ABB RobotStudio station: carsuspension.rspag

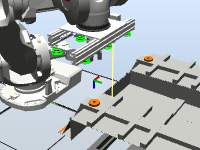
--- station ---
Station Car Suspension Ankit (saved by RobotStudio format 3)
Controller IRB_7600_340kg_2.80m
  mechanical unit ROB_1: IRB7600_340_280__01, 6 joints, base frame (0, 0, 0) mm
Layout (positions relative to the parent item):
  - IRB7600_340_280__01 [mechanism, from Robots\IRB7600_340_280_G_01.rslib] at (0, 0, 0) mm; joint values [1.0218, 0.5447, -0.711, 0.0026, 1.7386, 1.0222] (rad or m)
  - Part_10 [part, from Libraries\Part_10.rslib] at (-59.02, 745.49, 644.22) mm
  - SC_LaserSensor [smart component, from Libraries\SC_LaserSensor.rslib] at (1161.79, 1900.33, 1828.31) mm, rotated rx 180 ry -0.17 rz -180 deg
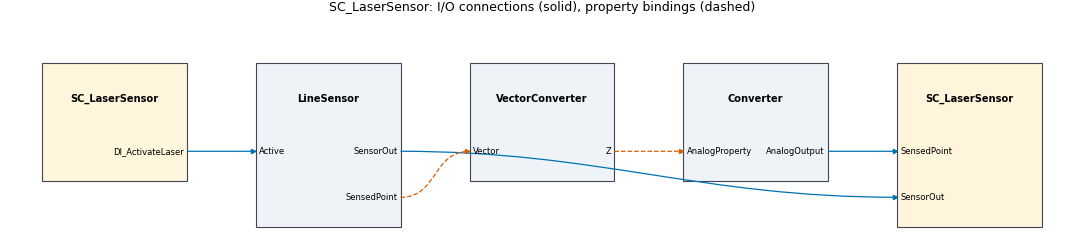
      connections:
        Converter.AnalogOutput -> SC_LaserSensor.SensedPoint
        LineSensor.SensorOut -> SC_LaserSensor.SensorOut
        SC_LaserSensor.DI_ActivateLaserSensor -> LineSensor.Active
        LineSensor.SensedPoint => VectorConverter.Vector
        VectorConverter.Z => Converter.AnalogProperty
    - LineSensor [smart component, from Components\LineSensor.rslib]
        properties: Start=[0.21 0.042 0.118]; End=[0.21 0.042 1]; Radius=1E-05; SensedPart=Car Underbody; SensedPoint=[0.949731506347656 1.94757446289063 1.11697045898437]
      - _sensorPart_ [part]
    - VectorConverter [smart component, from Components\VectorConverter.rslib]
        properties: X=0.949731506347656; Y=1.94757446289063; Z=1.11697045898437; Vector=[0.949731506347656 1.94757446289063 1.11697045898437]
    - Converter [smart component, from Components\Converter.rslib]
        properties: AnalogProperty=1.11697045898437; DigitalProperty=0; BooleanProperty=false; GroupProperty=0
  - table [part, from Libraries\table.rslib] at (1974.44, -431.38, 670) mm
  - Car Underbody [part] at (0, -200, 0) mm
  - SC_Gripper [smart component, from Libraries\SC_Gripper.rslib] at (-1443.39, 1900.33, 2562.23) mm, rotated rx 0 ry 60.17 rz 0 deg
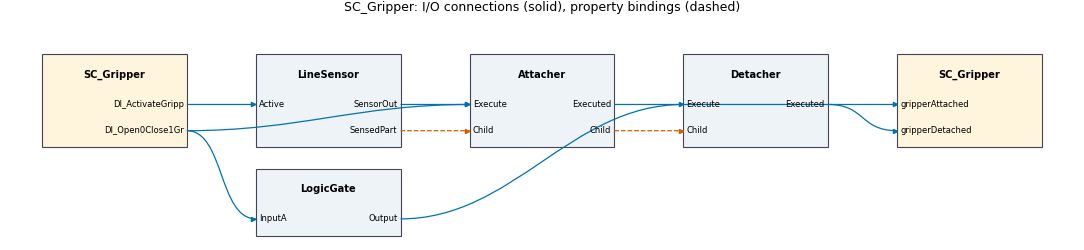
      connections:
        Attacher.Executed -> SC_Gripper.gripperAttached
        Detacher.Executed -> SC_Gripper.gripperDetached
        SC_Gripper.DI_ActivateGripper -> LineSensor.Active
        SC_Gripper.DI_Open0Close1Gripper -> Attacher.Execute
        LogicGate.Output -> Detacher.Execute
        SC_Gripper.DI_Open0Close1Gripper -> LogicGate.InputA
        LineSensor.SensorOut -> Attacher.Execute
        LineSensor.SensedPart => Attacher.Child
        Attacher.Child => Detacher.Child
    - Tool [graphiccomponentgroup, from Libraries\SC_Gripper.rslib] at (1932.51, 0, 1895) mm, rotated rx 180 ry 60 rz 180 deg
      - Vakuumgreifer [part, from Libraries\SC_Gripper.rslib]
      - GripperCylinder [part, from Libraries\SC_Gripper.rslib] at (0, 0, 85) mm
      - GripperFinger_1 [part, from Libraries\SC_Gripper.rslib] at (0, 0, 85) mm
      - GripperFinger_2 [part, from Libraries\SC_Gripper.rslib] at (0, 0, 85) mm, rotated rx 0 ry 0 rz 120 deg
      - GripperFinger_3 [part, from Libraries\SC_Gripper.rslib] at (0, 0, 85) mm, rotated rx 0 ry 0 rz -120 deg
    - LineSensor [smart component, from Components\LineSensor.rslib] at (1932.51, 0, 1895) mm, rotated rx 180 ry 60 rz 180 deg
        properties: Start=[0 0 0.215]; End=[0 0 0.225]; Radius=0.002; SensedPart=(none); SensedPoint=[1.29166296386719 1.83559130859375 1.60463647460938]
      - _sensorPart_ [part]
    - Attacher [smart component, from Components\Attacher.rslib]
        properties: Parent=Tool; Flange=0; Child=(none); Mount=false; Offset=[0 0 0]; Orientation=[0 0 0]
    - Detacher [smart component, from Components\Detacher.rslib]
        properties: Child=(none); KeepPosition=true
    - LogicGate [smart component, from Components\LogicGate.rslib]
        properties: Operator=NOT; Delay=0
  - Suspension_1 [graphiccomponentgroup, from Libraries\Suspension_1.rslib] at (2202.04, -555.68, 886.13) mm, rotated rx 180 ry 0 rz 0 deg
    - Part_4 [part, from Libraries\Suspension_1.rslib] at (0, 0, -2.49) mm
    - Part_5 [part, from Libraries\Suspension_1.rslib] at (0, 0, -2.05) mm
    - Part_6 [part, from Libraries\Suspension_1.rslib] at (0, 0, -2.05) mm
    - Part_3 [part, from Libraries\Suspension_1.rslib] at (-15.42, 2.83, 157.95) mm, rotated rx -180 ry 0 rz 0 deg
    - Part_7 [part, from Libraries\Suspension_1.rslib] at (15.59, 56.96, 120.72) mm, rotated rx -90 ry 0 rz -90 deg
  - Suspension_2 [graphiccomponentgroup, from Libraries\Suspension_2.rslib] at (2476.35, -555.68, 886.13) mm, rotated rx 180 ry 0 rz 0 deg
    - Part_4 [part, from Libraries\Suspension_2.rslib]
    - Part_5 [part, from Libraries\Suspension_2.rslib]
    - Part_6 [part, from Libraries\Suspension_2.rslib]
    - Part_3 [part, from Libraries\Suspension_2.rslib] at (-15.42, 2.83, 160) mm, rotated rx 180 ry 0 rz 0 deg
    - Part_7 [part, from Libraries\Suspension_2.rslib] at (15.59, 56.96, 122.77) mm, rotated rx -90 ry 0 rz -90 deg
Attachment: LineSensor is attached to Tool
Attachment: SC_Gripper is attached to IRB7600_340_280__01 / Link7
Attachment: Tool is attached to IRB7600_340_280__01 / Link7
Attachment: SC_LaserSensor is attached to IRB7600_340_280__01 / Link7
Attachment: Part_5 is attached to Part_4
Attachment: Part_6 is attached to Part_4
Attachment: Part_3 is attached to Part_4
Attachment: Part_7 is attached to Part_4
Attachment: Part_5 is attached to Part_4
Attachment: Part_6 is attached to Part_4
Attachment: Part_3 is attached to Part_4
Attachment: Part_7 is attached to Part_4
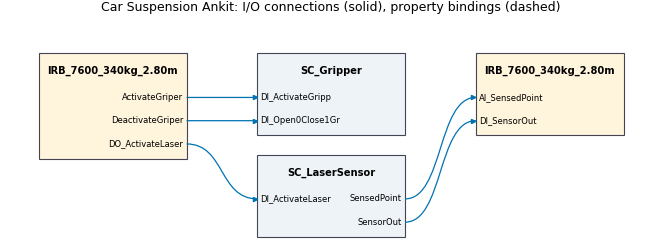
Station logic (signal -> signal, property => property):
  IRB_7600_340kg_2.80m.ActivateGriper -> SC_Gripper.DI_ActivateGripper
  IRB_7600_340kg_2.80m.DeactivateGriper -> SC_Gripper.DI_Open0Close1Gripper
  IRB_7600_340kg_2.80m.DO_ActivateLaserSensor -> SC_LaserSensor.DI_ActivateLaserSensor
  SC_LaserSensor.SensedPoint -> IRB_7600_340kg_2.80m.AI_SensedPoint
  SC_LaserSensor.SensorOut -> IRB_7600_340kg_2.80m.DI_SensorOut

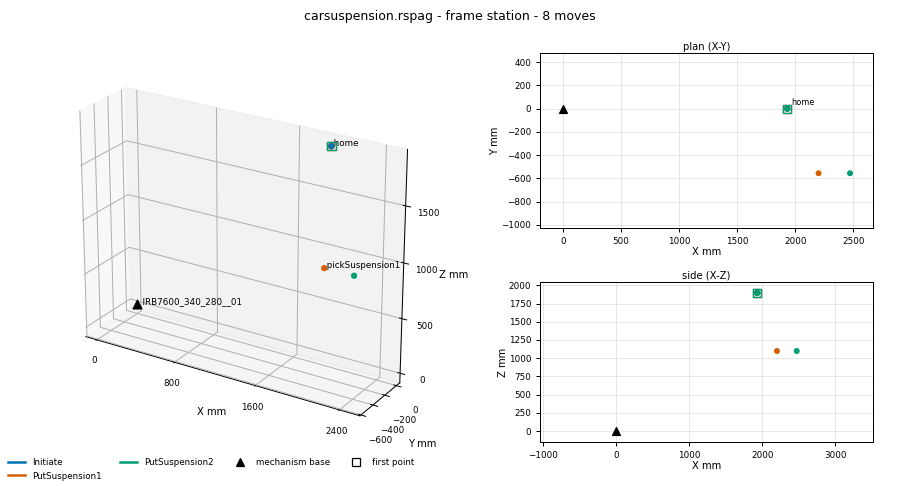
[picture p0: tool path of carsuspension.rspag in frame station, 8 of 38 moves have a stored position in this frame; points joined in program order, loops and branches not executed]
--- Backups/IRB_7600_340kg_2.80m/RAPID/TASK1/PROGMOD/CalibData.mod ---
MODULE CalibData
	TASK PERS tooldata myTool:=[TRUE,[[3.16,-2.44,456.26],[1,0,0,0]],[1,[0,0,1],[1,0,0,0],0,0,0]];
ENDMODULE

--- Backups/IRB_7600_340kg_2.80m/RAPID/TASK1/PROGMOD/Module1.mod ---
MODULE Module1
	CONST robtarget home:=[[1932.506319322,0,1894.999945226],[0.49999989,0,0.866025467,0],[0,0,0,0],[9E9,9E9,9E9,9E9,9E9,9E9]];
    CONST robtarget ScanFrontEdge:=[[201.51139568,1303.367736815,1894.998776679],[0.001498958,0.000001029,-0.999998877,0.000000047],[0,0,0,0],[9E9,9E9,9E9,9E9,9E9,9E9]];
    CONST robtarget pickSuspension1:=[[2201.608028845,-556.557878581,1098.980316128],[0.00023706,0.000000161,0.999999972,-0.00000152],[-1,0,-1,0],[9E9,9E9,9E9,9E9,9E9,9E9]];
    CONST robtarget pickSuspension2:=[[2472.738052401,-556.55975729,1098.980699702],[0.000237163,0.000000677,0.999999972,-0.000001447],[-1,0,-1,0],[9E9,9E9,9E9,9E9,9E9,9E9]];


    CONST num tcpYoffs:=42;
    CONST num tcpXoffs:=214.002;
    VAR robtarget Safehight;
    VAR robtarget next_target;
    VAR robtarget FrontEdge;
    VAR robtarget LeftEdge;
    VAR robtarget Centrep;
    VAR num HoleOffs;
    VAR robtarget CentrePoint1;
    VAR robtarget CentrePoint2;
    VAR robtarget CentrePoint3;
    VAR num Offsetz;
    VAR speeddata fast_speed:= v1000;
    VAR speeddata moderate_speed:= v500;


    PROC Initiate()
	    MoveJ home,fast_speed,z100,myTool\WObj:=wobj0;
        SetDO ActivateGriper,0;
        SetDO ActivateGriper,0;
        setdo DO_ActivateLaserSensor,0;
        Waitrob\InPos;
        WaitTime 1;
	ENDPROC

    PROC FrontEdge1()
        SetDO DO_ActivateLaserSensor,1;
        next_target:=ScanFrontEdge;

        MoveJ next_target,fast_speed,fine,tool0\WObj:=wobj0;
        WaitRob\InPos;
        WaitTime 1;
        WHILE TRUE DO
            IF  DI_SensorOut = 0 THEN
                next_target:=offs(next_target,0,100,0);
                MoveL next_target,fast_speed,fine,tool0\WObj:=wobj0;
                WaitRob\InPos;
                WaitTime 1;
            ELSE
                RETURN;
            ENDIF
        ENDWHILE
    ENDPROC
        PROC FrontEdge2()
            WHILE TRUE DO
                IF  DI_SensorOut = 1 THEN
                next_target:=Offs(next_target,0,-50,0);
                MoveL next_target,fast_speed,fine,tool0\WObj:=wobj0;
                WaitRob\InPos;
                WaitTime 0.1;
            ELSE
                FrontEdge:=next_target;
                RETURN;
                ENDIF
            ENDWHILE
        ENDPROC

         PROC FrontEdge3()
            WHILE TRUE DO
                IF  DI_SensorOut = 0 THEN
                next_target:=Offs(next_target,0,10,0);
                MoveL next_target,fast_speed,fine,tool0\WObj:=wobj0;
                WaitRob\InPos;
                WaitTime 0.1;
            ELSE
                FrontEdge:=next_target;
                RETURN;
                ENDIF
            ENDWHILE
        ENDPROC

         PROC FrontEdge4()
            WHILE TRUE DO
                IF  DI_SensorOut = 1 THEN
                next_target:=Offs(next_target,0,-1,0);
                MoveL next_target,fast_speed,fine,tool0\WObj:=wobj0;
                WaitRob\InPos;
                WaitTime 0.1;
            ELSE
                FrontEdge:=next_target;
                RETURN;
                ENDIF
            ENDWHILE
        ENDPROC

           PROC FrontEdge5()
            WHILE TRUE DO
                IF  DI_SensorOut = 0 THEN
                next_target:=Offs(next_target,0,0.1,0);
                MoveL next_target,fast_speed,fine,tool0\WObj:=wobj0;
                WaitRob\InPos;
                WaitTime 0.1;
            ELSE
                FrontEdge:=next_target;
                RETURN;
                ENDIF
            ENDWHILE
        ENDPROC

        PROC LeftEdge1()
            next_target:=Offs(FrontEdge,0,20,0);
            MoveL next_target,fast_speed,fine,tool0\WObj:=wobj0;
            WHILE TRUE DO
            IF   DI_SensorOut  = 1 THEN
                next_target:=Offs(next_target,-100,0,0);
                MoveL next_target,fast_speed,fine,tool0\WObj:=wobj0;
                WaitRob\InPos;
                WaitTime 0.5;
            ELSE
                RETURN;
            ENDIF
            ENDWHILE
        endproc
            PROC LeftEdge2()
                WHILE TRUE DO
                IF   DI_SensorOut  = 0 THEN
                next_target:=Offs(next_target,50,0,0);
                MoveL next_target,fast_speed,fine,tool0\WObj:=wobj0;
                ELSE
                LeftEdge:=Offs(next_target,-tcpXoffs,tcpYoffs,0);
                RETURN;
            ENDIF
                ENDWHILE
            ENDPROC

            PROC LeftEdge3()
                WHILE TRUE DO
                IF   DI_SensorOut  = 1 THEN
                next_target:=Offs(next_target,-10,0,0);
                MoveL next_target,fast_speed,fine,tool0\WObj:=wobj0;
                ELSE
                LeftEdge:=Offs(next_target,-tcpXoffs,tcpYoffs,0);
                RETURN;
            ENDIF
                ENDWHILE
            ENDPROC

             PROC LeftEdge4()
                WHILE TRUE DO
                IF   DI_SensorOut  = 0 THEN
                next_target:=Offs(next_target,1,0,0);
                MoveL next_target,fast_speed,fine,tool0\WObj:=wobj0;
                ELSE
                LeftEdge:=Offs(next_target,-tcpXoffs,tcpYoffs,0);
                RETURN;
            ENDIF
                ENDWHILE
            ENDPROC

             PROC LeftEdge5()
                WHILE TRUE DO
                IF   DI_SensorOut  = 1 THEN
                next_target:=Offs(next_target,-0.1,0,0);
                MoveL next_target,fast_speed,fine,tool0\WObj:=wobj0;
                ELSE
                LeftEdge:=Offs(next_target,-tcpXoffs,tcpYoffs,0);
                RETURN;
            ENDIF
                ENDWHILE
            ENDPROC


            PROC CentrePoint11()
                next_target:=Offs(next_target,220,150,0);
                MoveL next_target,fast_speed,fine,tool0\WObj:=wobj0;
                WHILE TRUE DO
                    IF  DI_SensorOut=1 THEN
                        next_target:=Offs(next_target,0,1,0);
                        MoveL next_target,fast_speed,fine,tool0\WObj:=wobj0;
                        WaitRob\InPos;
                        WaitTime 0.1;
                    ELSE
                        RETURN;
                    ENDIF
                ENDWHILE
            ENDPROC
            PROC CentrePoint12()
                 WHILE TRUE DO
                    IF  DI_SensorOut=0 THEN
                        next_target:=Offs(next_target,0,-0.1,0);
                        MoveL next_target,fast_speed,fine,tool0\WObj:=wobj0;
                        WaitRob\InPos;
                        WaitTime 0.1;
                    ELSE

                        CentrePoint1:=next_target;
                        RETURN;
                    ENDIF
                ENDWHILE
            ENDPROC
            PROC CentrePoint21()
                next_target:=Offs(next_target,0,1,0);
                MoveL next_target,fast_speed,fine,tool0\WObj:=wobj0;
                 WHILE TRUE DO
                    IF DI_Sensorout=0 THEN
                        next_target:=Offs(next_target,0,1,0);
                        MoveL next_target,fast_speed,fine,tool0\WObj:=wobj0;

                        WaitTime 1;
                    ELSE
                        Offsetz:=ai_Sensedpoint*1000;
                        RETURN;
                    ENDIF
                ENDWHILE
            ENDPROC
            PROC CentrePoint22()
                 WHILE TRUE DO
                    IF  DI_SensorOut=1 THEN
                        next_target:=Offs(next_target,0,-0.1,0);
                        MoveL next_target,fast_speed,fine,tool0\WObj:=wobj0;
                        WaitRob\InPos;
                        WaitTime 0.1;
                    ELSE

                        CentrePoint2:=next_target;
                        RETURN;
                    ENDIF
                ENDWHILE
            ENDPROC
            PROC CentrePoint31()
                 WHILE TRUE DO
                    IF  DI_SensorOut=0 THEN
                        next_target:=Offs(next_target,1,0,0);
                        MoveL next_target,fast_speed,fine,tool0\WObj:=wobj0;
                        WaitRob\InPos;
                        WaitTime 0.1;
                    ELSE
                        RETURN;
                    ENDIF
                ENDWHILE
            ENDPROC
            PROC CentrePoint32()
                 WHILE TRUE DO
                    IF  DI_SensorOut=1 THEN
                        next_target:=Offs(next_target,-0.1,0,0);
                        MoveL next_target,fast_speed,fine,tool0\WObj:=wobj0;
                        WaitRob\InPos;
                        WaitTime 0.1;
                    ELSE
                        CentrePoint3:=next_target;
                        RETURN;
                    ENDIF
                ENDWHILE
            ENDPROC
            PROC Centre()
                CentrePoint11;
                CentrePoint12;
                CentrePoint21;
                CentrePoint22;
                CentrePoint31;
                CentrePoint32;
                Centrep.trans.x:=(CentrePoint3.trans.x+CentrePoint1.trans.x)/2-tcpXoffs;
                Centrep.trans.y:=(CentrePoint3.trans.y+CentrePoint1.trans.y)/2+tcpYoffs;
                Centrep.trans.z:=Offsetz;
                Centrep.robconf:=CentrePoint3.robconf;
                Centrep.rot:=CentrePoint3.rot;
                Centrep.extax:=CentrePoint3.extax;
            ENDPROC

            PROC PutSuspension1()
                MoveL Home,fast_speed,fine,tool0\WObj:=wobj0;
                SafeHight:=Offs(pickSuspension1,0,0,500);
                MoveL Safehight,fast_speed,fine,tool0\WObj:=wobj0;
                MoveL pickSuspension1,fast_speed,fine,tool0\WObj:=wobj0;
                Setdo ActivateGriper,1;
                SetDO DeactivateGriper,1;
                WaitRob\InPos;
                WaitTime 0.5;
                MoveL Safehight,fast_speed,fine,tool0\WObj:=wobj0;
                MoveL Home,fast_speed,fine,tool0\WObj:=wobj0;
                Safehight:=offs(Centrep,0,0,250);
                MoveL Safehight,fast_speed,fine,myTool;
                MoveL Centrep,moderate_speed,fine,myTool;

                WaitRob\ZeroSpeed;
                 SetDO DeactivateGriper,0;
                MoveL Safehight,fast_speed,fine,myTool;
                SetDO ActivateGriper,0;
            ENDPROC

             PROC PutSuspension2()
                HoleOffs:=1430-(Centrep.trans.x-LeftEdge.trans.x)*2;
                MoveL Home,fast_speed,fine,tool0\WObj:=wobj0;
                Safehight:=Offs(pickSuspension2,0,0,200);
                MoveL Safehight,fast_speed,fine,tool0\WObj:=wobj0;
                MoveL pickSuspension2,fast_speed,fine,tool0\WObj:=wobj0;
                SetDO ActivateGriper,1;
                Setdo DeactivateGriper,1;
                WaitRob\InPos;
                WaitTime 0.5;
                MoveL Safehight,fast_speed,fine,tool0\WObj:=wobj0;
                SetDO ActivateGriper,0;
                MoveL Home,fast_speed,fine,tool0\WObj:=wobj0;

                MoveL Offs(Centrep,HoleOffs-8,0,200),fast_speed,fine,myTool;
                MoveL Offs(Centrep,HoleOffs-7,0,0),moderate_speed,fine,myTool;
                 WaitRob\ZeroSpeed;
                SetDO DeactivateGriper,0;

                Movej Offs(Centrep,HoleOffs-7,0,220),fast_speed,fine,myTool;
                SetDO ActivateGriper,0;
                MoveL Home,fast_speed,fine,tool0\WObj:=wobj0;
             ENDPROC



      PROC main()
        Initiate;
        FrontEdge1;
        FrontEdge2;
        FrontEdge3;
        FrontEdge4;
        FrontEdge5;
        LeftEdge1;
        LeftEdge2;
        LeftEdge3;
        LeftEdge4;
        LeftEdge5;
        Centre;
        PutSuspension1;
        PutSuspension2;

    ENDPROC

ENDMODULE

--- Backups/IRB_7600_340kg_2.80m/RAPID/TASK1/SYSMOD/LINKEDM.sys ---
%%%
  VERSION:1
  LANGUAGE:ENGLISH
%%%

MODULE LINKEDM (SYSMODULE)

! FOLLOWER
!     Name of electronically linked follower axis used by operator at teach pendent.
      PERS string l_f_axis_name{5}       :=  ["",  "", "", "", ""];

!     Name of the mechanical unit for follower axis.
      PERS string l_f_mecunt_n{5}  :=  ["", "", "", "", ""];

!     Linked follower axis number in the mechanical unit (first axis in mech. unit is number 1).
      PERS num l_f_axis_no{5}      :=  [0,          0,   0,  0,  0];

! MASTER
!     Name of the mechanical unit for linked master axis.
      PERS string l_m_mecunt_n{5} :=  ["", "", "", "", ""];

!     Linked master axis number in the mechanical unit (first axis in mech. unit is number 1).
!     See axis number table in documentation for different master mechanical units.
      PERS num l_m_axis_no{5}     :=  [0,  0,  0,  0,  0];

! POSITION OFFSET
!     The increase of the allowed offset position between the master and follower
!     positions, used when starting AUTO mode. As soon as the offset is decreased
!     the old configurated parameter is used.
!     Example: 3 => the configurated value of allowed offset is increased 3 times.
      PERS num offset_ratio{5}       :=  [10,  10,   10,  10,  10];

! SPEED RATIO
!     Speed_ratio used in AUTO and JOG modes [ very_slow   slow    normal    fast]
!     Value 1 = max allowed manual speed.
      CONST num speed_ratio {20}      := [0.01, 0.01, 0.01, 0.01, 0.01,
                                          0.05, 0.05, 0.05, 0.05, 0.05,
                                          0.20, 0.20, 0.20, 0.20, 0.20,
                                          1.00, 1.00, 1.00, 1.00, 1.00];

! STEP SIZE
!     Displacement position used in JOG mode for each activation of positive or
!     negative movement.                  [very_short    short   normal   long]
!     Unit degees or meter.
      CONST num displacement {20}     := [0.001, 0.001, 0.001, 0.001, 0.001,
                                          0.005, 0.005, 0.005, 0.005, 0.005,
                                          0.020, 0.020, 0.020, 0.020, 0.020,
                                          0.100, 0.100, 0.100, 0.100, 0.100];


!-------------------------------------------------------------
 PROC Linked_m ()
      Linked_m_exe ;
 ENDPROC
ENDMODULE

--- Backups/IRB_7600_340kg_2.80m/SYSPAR/EIO.cfg ---
EIO:CFG_1.0:6:1::
#
EIO_SIGNAL:

      -Name "DO_ActivateLaserSensor" -SignalType "DO" -Access "All"

      -Name "ActivateGriper" -SignalType "DO" -Access "All"

      -Name "DeactivateGriper" -SignalType "DO" -Access "All"

      -Name "DI_SensorOut" -SignalType "DI" -Access "All"

      -Name "AI_SensedPoint" -SignalType "AI" -Access "All"
